(*******************************************************************************
                          protoc-gen-twincat v0.0.0.0                           
             https://github.bhs-world.com/CorrML/protoc-gen-twincat             
*******************************************************************************)
{attribute 'no-analysis'}
TYPE ST_Bar :
STRUCT
	name : STRING;
	age : UDINT;
	email : STRING;
END_STRUCT
END_TYPE

(* stored: Version 1.1.0.1
   DUT ST_Bar: Id {0553817b-ed0a-4d2d-a69e-cd7a3638b266} *)
